Yaskawa INFORM job: REFPOINT_SERVO.JBI

/JOB
//NAME REFPOINT_SERVO
//POS
///NPOS 2,2,0,0,0,0
///TOOL 0
///POSTYPE PULSE
///PULSE
C00000=-91810,-61116,-26260,-36834,-11390,56133
C00001=-100924,20380,-44568,-6810,95866,-78623
BC00000=318426,679034,200539
BC00001=316385,679464,170794
//INST
///DATE 2025/04/16 15:02
///ATTR SC,RW
///GROUP1 RB1,BS1
NOP
MOVJ C00000 BC00000 VJ=5.00  //pkt1
MOVJ C00001 BC00001 VJ=5.00  //pkt2
END
